// TwinCAT 3 PLC project StructVarDemo
// ProgramVersion: 3.1.4023.0
// libraries:
//   Tc2_Standard, * (Beckhoff Automation GmbH)
//   Tc2_System, * (Beckhoff Automation GmbH)
//   Tc3_Module, * (Beckhoff Automation GmbH)
// project tree:
//   DUTs/ MotorVariables.TcDUT
//   / PlcTask.TcTTO
//   POUs/ MAIN.TcPOU, Motor.TcPOU, Plc_Prog.TcPOU
// real-time tasks:
//   TASK PlcTask: cycle T#10ms, priority 20, ADS port 350

CONFIGURATION StructVarDemo
    RESOURCE PLC ON TwinCAT3
        TASK PlcTask(INTERVAL := T#10ms, PRIORITY := 20);
        PROGRAM MAIN WITH PlcTask : MAIN;
    END_RESOURCE
END_CONFIGURATION

// ---- DUTs/MotorVariables.TcDUT
TYPE MotorVariables :
STRUCT
	Start : BOOL;
	Stop : BOOL;
	Oveload : BOOL;
	Coil : BOOL;
	
END_STRUCT
END_TYPE

// ---- POUs/MAIN.TcPOU
PROGRAM MAIN
VAR
END_VAR

Plc_Prog();

END_PROGRAM

// ---- POUs/Plc_Prog.TcPOU
PROGRAM Plc_Prog
VAR
	Motor1 : Motor;
	Motor2 : Motor;
	Motor3 : Motor;
	
	Motor1Variables : MotorVariables;
	Motor2Variables : MotorVariables;
	Motor3Variables : MotorVariables;
END_VAR

Motor1(Start:=Motor1Variables.Start, Stop:=Motor1Variables.Stop, Overload:=Motor1Variables.Oveload, Coil=>Motor1Variables.Coil);
Motor2(Start:=Motor2Variables.Start, Stop:=Motor2Variables.Stop, Overload:=Motor2Variables.Oveload, Coil=>Motor2Variables.Coil);
Motor3(Start:=Motor3Variables.Start, Stop:=Motor3Variables.Stop, Overload:=Motor3Variables.Oveload, Coil=>Motor3Variables.Coil);

END_PROGRAM

// ---- POUs/Motor.TcPOU
FUNCTION_BLOCK Motor
VAR_INPUT
	Start: BOOL;
	Stop : BOOL;
	Overload : BOOL;
END_VAR
VAR_OUTPUT
	Coil : BOOL;
END_VAR
VAR
END_VAR

IF Start AND Stop = FALSE AND Overload = FALSE THEN
	Coil := TRUE;
ELSE
	Coil := FALSE;
	
END_IF

END_FUNCTION_BLOCK
